Staubli VAL3: exePulse.pgx

program exePulse(dio x_dDio, num x_nLength)
begin

  //pulse execution

  x_dDio=true
  delay(x_nLength)
  x_dDio=false

end
